Staubli VAL3: buildList.pgx

program buildList()
  local num l_nSize
  local string l_sEvent
  local num i
  local bool l_bFound
  local num l_nCount
  local string l_sEmpty
begin
  // INIT the list
  l_sEmpty=""
  call use:stringCopy(l_sEmpty,sList)
  // Build the list
  call trajType:getSize(l_nSize)
  for i=0 to l_nSize-1
    call trajType:get(l_sEvent,i)
    if l_sEvent!=""
      //
      // use the filter ?
      //
      // check if the bProcessList filter is active
      //
      l_bFound=true
      if saveData:sTrajFilter!=""
        l_bFound=find(l_sEvent,saveData:sTrajFilter)!=-1
      endIf
      // update the selected item
      if l_sEvent==sEvent
        nSelected=l_nCount
      endIf
      // add
      if l_bFound
        call listAdd(l_sEvent)
        l_nCount=l_nCount+1
      endIf
    endIf
  endFor
  // update
  use:bUseRefresh=true
end
